// TIA Portal V21 export
FUNCTION_BLOCK "MotorSoftstart"   // FB8889, LAD
{ S7_Optimized_Access := 'TRUE' }
// stored: AutoNumber false, MemoryReserve 100, SetENOAutomatically false
   VAR_INPUT
      FI_AutoConditions { ExternalAccessible := 'False'; ExternalVisible := 'False'; ExternalWritable := 'False'} : Bool;
      FI_AutoForward { ExternalAccessible := 'False'; ExternalVisible := 'False'; ExternalWritable := 'False'} : Bool;
      FI_ProfinetOK { ExternalAccessible := 'False'; ExternalVisible := 'False'; ExternalWritable := 'False'} : Bool;
      FI_CircuitProtectionOK { ExternalAccessible := 'False'; ExternalVisible := 'False'; ExternalWritable := 'False'} : Bool;
      FI_SoftstartAlarm { ExternalAccessible := 'False'; ExternalVisible := 'False'; ExternalWritable := 'False'} : Bool;
      FI_ContactorON { ExternalAccessible := 'False'; ExternalVisible := 'False'; ExternalWritable := 'False'} : Bool;
      FI_SoftstartON { ExternalAccessible := 'False'; ExternalVisible := 'False'; ExternalWritable := 'False'} : Bool;
      FI_SoftstartBypassed { ExternalAccessible := 'False'; ExternalVisible := 'False'; ExternalWritable := 'False'} : Bool;
      FI_ManualMode { ExternalAccessible := 'False'; ExternalVisible := 'False'; ExternalWritable := 'False'} : Bool;
      FI_EmergencyStop { ExternalAccessible := 'False'; ExternalVisible := 'False'; ExternalWritable := 'False'} : Bool;
      FI_Reset { ExternalAccessible := 'False'; ExternalVisible := 'False'; ExternalWritable := 'False'} : Bool;
   END_VAR
   VAR_OUTPUT
      FQ_ContactorON { ExternalAccessible := 'False'; ExternalVisible := 'False'; ExternalWritable := 'False'} : Bool;
      FQ_MotorStart { ExternalAccessible := 'False'; ExternalVisible := 'False'; ExternalWritable := 'False'} : Bool;
      FQ_AlarmCircuitProtection { ExternalAccessible := 'False'; ExternalVisible := 'False'; ExternalWritable := 'False'} : Bool;
      FQ_AlarmContactorNotON { ExternalAccessible := 'False'; ExternalVisible := 'False'; ExternalWritable := 'False'} : Bool;
      FQ_AlarmContactorNotOFF { ExternalAccessible := 'False'; ExternalVisible := 'False'; ExternalWritable := 'False'} : Bool;
      FQ_AlarmSoftstartNotON { ExternalAccessible := 'False'; ExternalVisible := 'False'; ExternalWritable := 'False'} : Bool;
      FQ_AlarmSoftstartNotBypassed { ExternalAccessible := 'False'; ExternalVisible := 'False'; ExternalWritable := 'False'} : Bool;
      FQ_AlarmSoftstartStuckBypassed { ExternalAccessible := 'False'; ExternalVisible := 'False'; ExternalWritable := 'False'} : Bool;
      FQ_AlarmSoftstartNotOFF { ExternalAccessible := 'False'; ExternalVisible := 'False'; ExternalWritable := 'False'} : Bool;
      FQ_AlarmSoftstartFault { ExternalAccessible := 'False'; ExternalVisible := 'False'; ExternalWritable := 'False'} : Bool;
   END_VAR
   VAR_IN_OUT
      FIQ_WorkTime : "UDT_WORK_CNT";
      FIQ_DeviceState : "UDT_Device";
   END_VAR
   VAR
      generalConditions { ExternalAccessible := 'False'; ExternalVisible := 'False'; ExternalWritable := 'False'} : Bool;
      Authorisation { ExternalAccessible := 'False'; ExternalVisible := 'False'; ExternalWritable := 'False'} : Bool;
      Alarm { ExternalAccessible := 'False'; ExternalVisible := 'False'; ExternalWritable := 'False'} : Bool;
      contactorON { ExternalAccessible := 'False'; ExternalVisible := 'False'; ExternalWritable := 'False'} : Bool;
      motorStart { ExternalAccessible := 'False'; ExternalVisible := 'False'; ExternalWritable := 'False'} : Bool;
      motorConfirmed { ExternalAccessible := 'False'; ExternalVisible := 'False'; ExternalWritable := 'False'} : Bool;
      Timers { ExternalAccessible := 'False'; ExternalVisible := 'False'; ExternalWritable := 'False'} : Struct
         CircuitProtection : TON_TIME;
         ContNotON : TON_TIME;
         ContNotOFF : TON_TIME;
         SoftstartNotON : TON_TIME;
         SoftstartNotOFF : TON_TIME;
         SoftstartNotBypassed : TON_TIME;
         SoftstartBypassed : TON_TIME;
         SoftstartFailure : TON_TIME;
      END_STRUCT;
      C_WORK_TIME { ExternalAccessible := 'False'; ExternalVisible := 'False'; ExternalWritable := 'False'} : "TIME_COUNTER_FB";
   END_VAR
BEGIN

REGION Network 1: General conditions
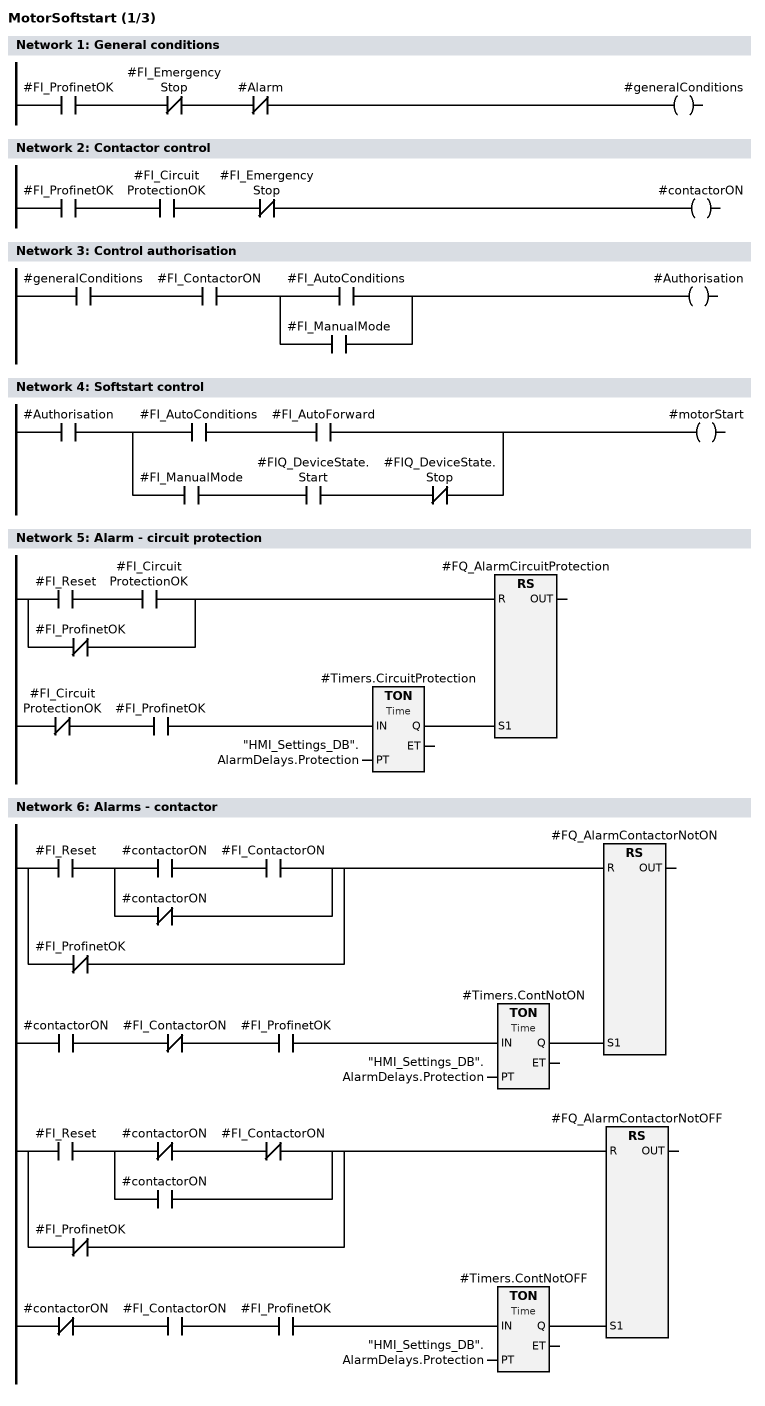
   RUNG wire#powerrail
      Contact( #FI_ProfinetOK )
      I_Contact( #FI_EmergencyStop )
      I_Contact( #Alarm )
      Coil( #generalConditions )
   END_RUNG
   // the same network as SCL:
   #generalConditions := #FI_ProfinetOK AND NOT #FI_EmergencyStop AND NOT #Alarm;
END_REGION

REGION Network 2: Contactor control
   RUNG wire#powerrail
      Contact( #FI_ProfinetOK )
      Contact( #FI_CircuitProtectionOK )
      I_Contact( #FI_EmergencyStop )
      Coil( #contactorON )
   END_RUNG
   // the same network as SCL:
   #contactorON := #FI_ProfinetOK AND #FI_CircuitProtectionOK AND NOT #FI_EmergencyStop;
END_REGION

REGION Network 3: Control authorisation
   RUNG wire#powerrail
      Contact( #generalConditions )
      Contact( #FI_ContactorON )
      wire#w1
      Contact( #FI_AutoConditions )
      wire#w2
      Coil( #Authorisation )
   END_RUNG
   RUNG wire#w1
      Contact( #FI_ManualMode )
   END_RUNG wire#w2
   // the same network as SCL:
   #Authorisation := #generalConditions AND #FI_ContactorON AND (#FI_AutoConditions OR #FI_ManualMode);
END_REGION

REGION Network 4: Softstart control
   RUNG wire#powerrail
      Contact( #Authorisation )
      wire#w1
      Contact( #FI_AutoConditions )
      Contact( #FI_AutoForward )
      wire#w2
      Coil( #motorStart )
   END_RUNG
   RUNG wire#w1
      Contact( #FI_ManualMode )
      Contact( #FIQ_DeviceState.Start )
      I_Contact( #FIQ_DeviceState.Stop )
   END_RUNG wire#w2
   // the same network as SCL:
   #motorStart := #Authorisation AND ((#FI_AutoConditions AND #FI_AutoForward) OR (#FI_ManualMode AND #FIQ_DeviceState.Start AND NOT #FIQ_DeviceState.Stop));
END_REGION

REGION Network 5: Alarm - circuit protection
   RUNG wire#powerrail
      Contact( #FI_Reset )
      Contact( #FI_CircuitProtectionOK )
      wire#w1
      S_RS(operand := #FQ_AlarmCircuitProtection, s1 := wire#w2)
   END_RUNG
   RUNG wire#powerrail
      I_Contact( #FI_ProfinetOK )
   END_RUNG wire#w1
   RUNG wire#powerrail
      I_Contact( #FI_CircuitProtectionOK )
      Contact( #FI_ProfinetOK )
      { S7_Templates := "time_type := Time" } #Timers.CircuitProtection.TON(pt := "HMI_Settings_DB".AlarmDelays.Protection, et =>)
   END_RUNG wire#w2
   // the same network as SCL:
   #Timers.CircuitProtection.TON(IN := NOT #FI_CircuitProtectionOK AND #FI_ProfinetOK,
                           PT := "HMI_Settings_DB".AlarmDelays.Protection);
   IF (#FI_Reset AND #FI_CircuitProtectionOK) OR NOT #FI_ProfinetOK THEN
       #FQ_AlarmCircuitProtection := FALSE;   // RS flip-flop
   END_IF;
   IF #Timers.CircuitProtection.Q THEN #FQ_AlarmCircuitProtection := TRUE; END_IF;
END_REGION

REGION Network 6: Alarms - contactor
   RUNG wire#powerrail
      Contact( #FI_Reset )
      wire#w1
      Contact( #contactorON )
      Contact( #FI_ContactorON )
      wire#w2
      S_RS(operand := #FQ_AlarmContactorNotON, s1 := wire#w3)
   END_RUNG
   RUNG wire#w1
      I_Contact( #contactorON )
   END_RUNG wire#w2
   RUNG wire#powerrail
      I_Contact( #FI_ProfinetOK )
   END_RUNG wire#w2
   RUNG wire#powerrail
      Contact( #contactorON )
      I_Contact( #FI_ContactorON )
      Contact( #FI_ProfinetOK )
      { S7_Templates := "time_type := Time" } #Timers.ContNotON.TON(pt := "HMI_Settings_DB".AlarmDelays.Protection, et =>)
   END_RUNG wire#w3
   RUNG wire#powerrail
      Contact( #FI_Reset )
      wire#w4
      I_Contact( #contactorON )
      I_Contact( #FI_ContactorON )
      wire#w5
      S_RS(operand := #FQ_AlarmContactorNotOFF, s1 := wire#w6)
   END_RUNG
   RUNG wire#w4
      Contact( #contactorON )
   END_RUNG wire#w5
   RUNG wire#powerrail
      I_Contact( #FI_ProfinetOK )
   END_RUNG wire#w5
   RUNG wire#powerrail
      I_Contact( #contactorON )
      Contact( #FI_ContactorON )
      Contact( #FI_ProfinetOK )
      { S7_Templates := "time_type := Time" } #Timers.ContNotOFF.TON(pt := "HMI_Settings_DB".AlarmDelays.Protection, et =>)
   END_RUNG wire#w6
   // the same network as SCL:
   #Timers.ContNotON.TON(IN := #contactorON AND NOT #FI_ContactorON AND #FI_ProfinetOK,
                         PT := "HMI_Settings_DB".AlarmDelays.Protection);
   IF (#FI_Reset AND ((#contactorON AND #FI_ContactorON) OR NOT #contactorON)) OR NOT #FI_ProfinetOK THEN
       #FQ_AlarmContactorNotON := FALSE;   // RS flip-flop
   END_IF;
   IF #Timers.ContNotON.Q THEN #FQ_AlarmContactorNotON := TRUE; END_IF;
   #Timers.ContNotOFF.TON(IN := NOT #contactorON AND #FI_ContactorON AND #FI_ProfinetOK,
                          PT := "HMI_Settings_DB".AlarmDelays.Protection);
   IF (#FI_Reset AND ((NOT #contactorON AND NOT #FI_ContactorON) OR #contactorON)) OR NOT #FI_ProfinetOK THEN
       #FQ_AlarmContactorNotOFF := FALSE;   // RS flip-flop
   END_IF;
   IF #Timers.ContNotOFF.Q THEN #FQ_AlarmContactorNotOFF := TRUE; END_IF;
END_REGION

REGION Network 7: Alarm - softstart not ON
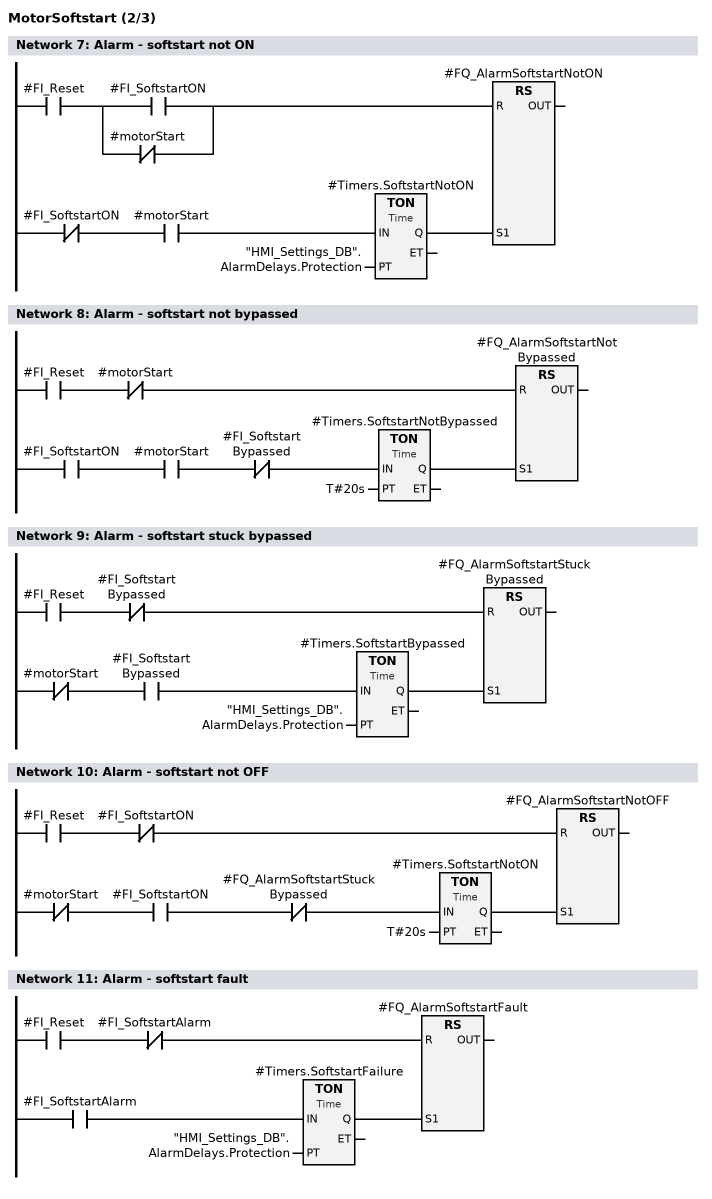
   RUNG wire#powerrail
      Contact( #FI_Reset )
      wire#w1
      Contact( #FI_SoftstartON )
      wire#w2
      S_RS(operand := #FQ_AlarmSoftstartNotON, s1 := wire#w3)
   END_RUNG
   RUNG wire#w1
      I_Contact( #motorStart )
   END_RUNG wire#w2
   RUNG wire#powerrail
      I_Contact( #FI_SoftstartON )
      Contact( #motorStart )
      { S7_Templates := "time_type := Time" } #Timers.SoftstartNotON.TON(pt := "HMI_Settings_DB".AlarmDelays.Protection, et =>)
   END_RUNG wire#w3
   // the same network as SCL:
   #Timers.SoftstartNotON.TON(IN := NOT #FI_SoftstartON AND #motorStart,
                           PT := "HMI_Settings_DB".AlarmDelays.Protection);
   IF #FI_Reset AND (#FI_SoftstartON OR NOT #motorStart) THEN
       #FQ_AlarmSoftstartNotON := FALSE;   // RS flip-flop
   END_IF;
   IF #Timers.SoftstartNotON.Q THEN #FQ_AlarmSoftstartNotON := TRUE; END_IF;
END_REGION

REGION Network 8: Alarm - softstart not bypassed
   RUNG wire#powerrail
      Contact( #FI_Reset )
      I_Contact( #motorStart )
      S_RS(operand := #FQ_AlarmSoftstartNotBypassed, s1 := wire#w1)
   END_RUNG
   RUNG wire#powerrail
      Contact( #FI_SoftstartON )
      Contact( #motorStart )
      I_Contact( #FI_SoftstartBypassed )
      { S7_Templates := "time_type := Time" } #Timers.SoftstartNotBypassed.TON(pt := T#20s, et =>)
   END_RUNG wire#w1
   // the same network as SCL:
   #Timers.SoftstartNotBypassed.TON(IN := #FI_SoftstartON AND #motorStart AND NOT #FI_SoftstartBypassed,
                           PT := T#20s);
   IF #FI_Reset AND NOT #motorStart THEN
       #FQ_AlarmSoftstartNotBypassed := FALSE;   // RS flip-flop
   END_IF;
   IF #Timers.SoftstartNotBypassed.Q THEN #FQ_AlarmSoftstartNotBypassed := TRUE; END_IF;
END_REGION

REGION Network 9: Alarm - softstart stuck bypassed
   RUNG wire#powerrail
      Contact( #FI_Reset )
      I_Contact( #FI_SoftstartBypassed )
      S_RS(operand := #FQ_AlarmSoftstartStuckBypassed, s1 := wire#w1)
   END_RUNG
   RUNG wire#powerrail
      I_Contact( #motorStart )
      Contact( #FI_SoftstartBypassed )
      { S7_Templates := "time_type := Time" } #Timers.SoftstartBypassed.TON(pt := "HMI_Settings_DB".AlarmDelays.Protection, et =>)
   END_RUNG wire#w1
   // the same network as SCL:
   #Timers.SoftstartBypassed.TON(IN := NOT #motorStart AND #FI_SoftstartBypassed,
                           PT := "HMI_Settings_DB".AlarmDelays.Protection);
   IF #FI_Reset AND NOT #FI_SoftstartBypassed THEN
       #FQ_AlarmSoftstartStuckBypassed := FALSE;   // RS flip-flop
   END_IF;
   IF #Timers.SoftstartBypassed.Q THEN #FQ_AlarmSoftstartStuckBypassed := TRUE; END_IF;
END_REGION

REGION Network 10: Alarm - softstart not OFF
   RUNG wire#powerrail
      Contact( #FI_Reset )
      I_Contact( #FI_SoftstartON )
      S_RS(operand := #FQ_AlarmSoftstartNotOFF, s1 := wire#w1)
   END_RUNG
   RUNG wire#powerrail
      I_Contact( #motorStart )
      Contact( #FI_SoftstartON )
      I_Contact( #FQ_AlarmSoftstartStuckBypassed )
      { S7_Templates := "time_type := Time" } #Timers.SoftstartNotON.TON(pt := T#20s, et =>)
   END_RUNG wire#w1
   // the same network as SCL:
   #Timers.SoftstartNotON.TON(IN := NOT #motorStart AND #FI_SoftstartON AND NOT #FQ_AlarmSoftstartStuckBypassed,
                           PT := T#20s);
   IF #FI_Reset AND NOT #FI_SoftstartON THEN
       #FQ_AlarmSoftstartNotOFF := FALSE;   // RS flip-flop
   END_IF;
   IF #Timers.SoftstartNotON.Q THEN #FQ_AlarmSoftstartNotOFF := TRUE; END_IF;
END_REGION

REGION Network 11: Alarm - softstart fault
   RUNG wire#powerrail
      Contact( #FI_Reset )
      I_Contact( #FI_SoftstartAlarm )
      S_RS(operand := #FQ_AlarmSoftstartFault, s1 := wire#w1)
   END_RUNG
   RUNG wire#powerrail
      Contact( #FI_SoftstartAlarm )
      { S7_Templates := "time_type := Time" } #Timers.SoftstartFailure.TON(pt := "HMI_Settings_DB".AlarmDelays.Protection, et =>)
   END_RUNG wire#w1
   // the same network as SCL:
   #Timers.SoftstartFailure.TON(IN := #FI_SoftstartAlarm, PT := "HMI_Settings_DB".AlarmDelays.Protection);
   IF #FI_Reset AND NOT #FI_SoftstartAlarm THEN
       #FQ_AlarmSoftstartFault := FALSE;   // RS flip-flop
   END_IF;
   IF #Timers.SoftstartFailure.Q THEN #FQ_AlarmSoftstartFault := TRUE; END_IF;
END_REGION

REGION Network 12: Any alarm
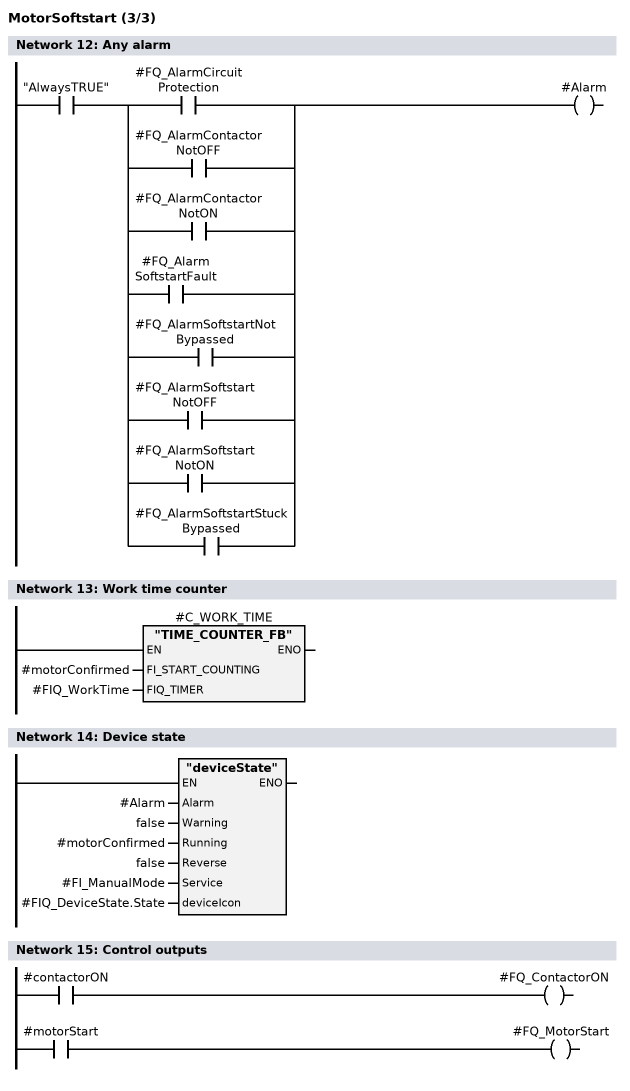
   RUNG wire#powerrail
      Contact( "AlwaysTRUE" )
      wire#w1
      Contact( #FQ_AlarmCircuitProtection )
      wire#w2
      Coil( #Alarm )
   END_RUNG
   RUNG wire#w1
      Contact( #FQ_AlarmContactorNotOFF )
   END_RUNG wire#w2
   RUNG wire#w1
      Contact( #FQ_AlarmContactorNotON )
   END_RUNG wire#w2
   RUNG wire#w1
      Contact( #FQ_AlarmSoftstartFault )
   END_RUNG wire#w2
   RUNG wire#w1
      Contact( #FQ_AlarmSoftstartNotBypassed )
   END_RUNG wire#w2
   RUNG wire#w1
      Contact( #FQ_AlarmSoftstartNotOFF )
   END_RUNG wire#w2
   RUNG wire#w1
      Contact( #FQ_AlarmSoftstartNotON )
   END_RUNG wire#w2
   RUNG wire#w1
      Contact( #FQ_AlarmSoftstartStuckBypassed )
   END_RUNG wire#w2
   // the same network as SCL:
   #Alarm := "AlwaysTRUE" AND (#FQ_AlarmCircuitProtection OR #FQ_AlarmContactorNotOFF OR #FQ_AlarmContactorNotON OR #FQ_AlarmSoftstartFault OR #FQ_AlarmSoftstartNotBypassed OR #FQ_AlarmSoftstartNotOFF OR #FQ_AlarmSoftstartNotON OR #FQ_AlarmSoftstartStuckBypassed);
END_REGION

REGION Network 13: Work time counter
   RUNG wire#powerrail
      #C_WORK_TIME(FI_START_COUNTING := #motorConfirmed, FIQ_TIMER := #FIQ_WorkTime)
   END_RUNG
   // the same network as SCL:
   #C_WORK_TIME(FI_START_COUNTING := #motorConfirmed, FIQ_TIMER := #FIQ_WorkTime);   // "TIME_COUNTER_FB"
END_REGION

REGION Network 14: Device state
   RUNG wire#powerrail
      "deviceState"(Alarm := #Alarm, Warning := false, Running := #motorConfirmed, Reverse := false, Service := #FI_ManualMode, deviceIcon := #FIQ_DeviceState.State)
   END_RUNG
   // the same network as SCL:
   "deviceState"(Alarm := #Alarm,
                 Warning := false,
                 Running := #motorConfirmed,
                 Reverse := false,
                 Service := #FI_ManualMode,
                 deviceIcon := #FIQ_DeviceState.State);
END_REGION

REGION Network 15: Control outputs
   RUNG wire#powerrail
      Contact( #contactorON )
      Coil( #FQ_ContactorON )
   END_RUNG
   RUNG wire#powerrail
      Contact( #motorStart )
      Coil( #FQ_MotorStart )
   END_RUNG
   // the same network as SCL:
   #FQ_ContactorON := #contactorON;
   #FQ_MotorStart := #motorStart;
END_REGION
END_FUNCTION_BLOCK
